(* PLC project  *)

PROGRAM P
  VAR
    fb : FB_Buf;
  END_VAR

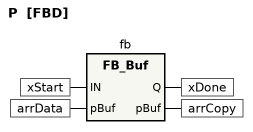
(* FBD diagram, written out as Structured Text *)
fb(IN := xStart, pBuf := arrData);
xDone := fb.Q;
arrCopy := fb.pBuf;
END_PROGRAM
